FUNCTION_BLOCK FB_CalcImageDistance
VAR_INPUT
END_VAR
VAR_OUTPUT
END_VAR
VAR
END_VAR

END_FUNCTION_BLOCK

(* stored: Version 1.1.0.1, ProductVersion 3.1.4022.18
   POU FB_CalcImageDistance: Id {81fe0328-7a74-4932-bc70-1630590071fc}, SpecialFunc None *)
